FUNCTION_BLOCK DelayedActive (* Composite Function Block Type *)
  (* Standard: 61499-2 *)
  (* Version 0.0, 6/19/2026, Schneider Electric, template *)
  PACKAGE SE.Nereda;
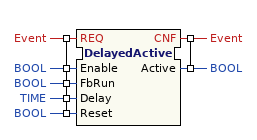
  EVENT_INPUT
    REQ WITH FbRun, Delay, Reset, Enable;
  END_EVENT
  EVENT_OUTPUT
    CNF WITH Active; (* Execution Confirmation *)
  END_EVENT
  VAR_INPUT
    Enable : BOOL;
    FbRun : BOOL;
    Delay : TIME; (* Delay Time *)
    Reset : BOOL;
  END_VAR
  VAR_OUTPUT
    Active : BOOL;
  END_VAR
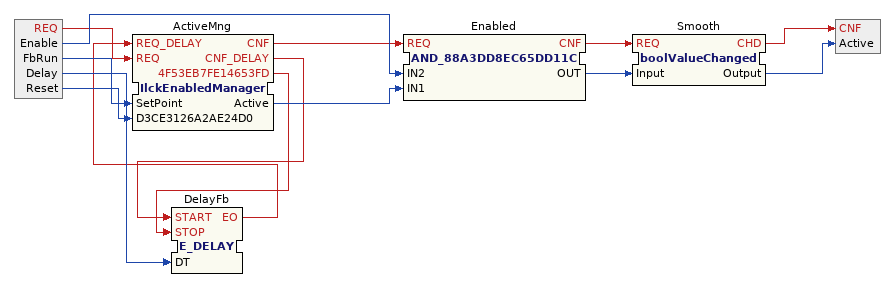
  FBS
    ActiveMng : IlckEnabledManager;
    DelayFb : E_DELAY;
    Smooth : boolValueChanged;
    Enabled : AND_88A3DD8EC65DD11C; {SET_ATTRIBUTE(Configuration.GenericFBType.InterfaceParams, Runtime.Standard#CNT:=2;OUT:BOOL)}
  END_FBS
  EVENT_CONNECTIONS
    Smooth.CHD TO CNF;
    Enabled.CNF TO Smooth.REQ;
    ActiveMng.CNF TO Enabled.REQ;
    ActiveMng.CNF_DELAY TO DelayFb.START;
    DelayFb.EO TO ActiveMng.REQ_DELAY;
    REQ TO ActiveMng.REQ;
    ActiveMng.4F53EB7FE14653FD TO DelayFb.STOP;
  END_CONNECTIONS
  DATA_CONNECTIONS
    Delay TO DelayFb.DT;
    Smooth.Output TO Active;
    Enabled.OUT TO Smooth.Input;
    Enable TO Enabled.IN2;
    ActiveMng.Active TO Enabled.IN1;
    FbRun TO ActiveMng.SetPoint;
    Reset TO ActiveMng.D3CE3126A2AE24D0;
  END_CONNECTIONS
END_FUNCTION_BLOCK
